// TIA Portal V18 export
FUNCTION_BLOCK "SCALING"   // FB4, LAD
{ S7_Optimized_Access := 'TRUE' }
VERSION : 0.1
// stored: AutoNumber true, IsIECCheckEnabled false, IsRetainMemResEnabled false, MemoryReserve 100, SetENOAutomatically false, UDAEnableTagReadback false
   VAR_INPUT
      RAW_MIN : Int;
      RAW_MAX : Int;
      INPUT : Int;
      SCALE_MIN : Real;
      SCALE_MAX : Real;
   END_VAR
   VAR_OUTPUT
      SCALE_OUT : Real;
   END_VAR
   VAR
      TEMP : Real;
   END_VAR
BEGIN

REGION Network 1: SCALING_BLOCK
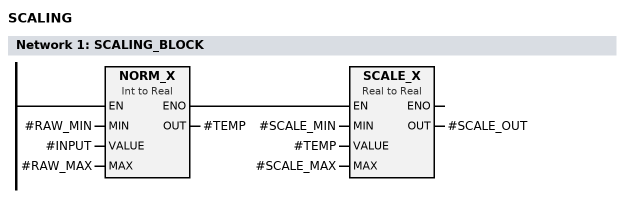
   RUNG wire#powerrail
      { S7_Templates := "[SrcType := Int, DestType := Real]" } Normalize(min := #RAW_MIN, value := #INPUT, max := #RAW_MAX, out => #TEMP)
      { S7_Templates := "[SrcType := Real, DestType := Real]" } Scale(min := #SCALE_MIN, value := #TEMP, max := #SCALE_MAX, out => #SCALE_OUT)
   END_RUNG
   // the same network as SCL:
   #TEMP := NORM_X(MIN := #RAW_MIN, VALUE := #INPUT, MAX := #RAW_MAX);
   #SCALE_OUT := SCALE_X(MIN := #SCALE_MIN, VALUE := #TEMP, MAX := #SCALE_MAX);
END_REGION
END_FUNCTION_BLOCK
